{attribute 'GeneratedUsingTerminal: EL6001-0000-0020'}
{attribute addProperty BoxType "EL6001-0000-0020"}
{attribute addProperty Id "COM_ext_inputsAT %I*COM_ext_inputs_1F197B20108COM_ext_outputsAT %Q*COM_ext_outputs_54D54ACC105WcStateAT %I*WcState_9091E0EB2InfoDataAT %I*InfoData_32EB74EA10"}
{attribute addProperty CRC "4118337059"}
{attribute addProperty Size "225"}
TYPE EL6001_F578D623 EXTENDS EtcSlaveTerminalBase_947E5A46 :
STRUCT
	{attribute addProperty Name "COM_ext_inputs"}
	COM_ext_inputs : COM_ext_inputs_1F197B20;
	{attribute addProperty Name "COM_ext_outputs"}
	COM_ext_outputs : COM_ext_outputs_54D54ACC;
	{attribute addProperty Name "WcState"}
	WcState : WcState_9091E0EB;
	{attribute addProperty Name "InfoData"}
	InfoData : InfoData_32EB74EA;
END_STRUCT
END_TYPE

(* stored: Version 1.2.0.0, ProductVersion 3.1.4024.9
   DUT EL6001_F578D623: Id {f6ab5357-6265-439b-8112-e922d57c4771} *)
